{attribute 'linkalways'} 
{attribute 'no_explicit_call' := 'This FB is a CLASS and must be accessed using methods or properties'}
{attribute 'enable_dynamic_creation'}
FUNCTION_BLOCK Node_F_VN_BoxFilter EXTENDS VisionNode
VAR
	ipSrcImage : _ITcVnImage;
    ipDestImage : _ITcVnImage;
    nFilterWidth : _UDINT(1);
    nFilterHeight : _UDINT(1);
    hrPrev : _HRESULT(S_OK);
	hresult : _HRESULT(S_OK);
END_VAR

METHOD PUBLIC  Clone : I_Node
VAR
	pNode : POINTER TO Node_F_VN_BoxFilter;
END_VAR
pNode := __NEW(Node_F_VN_BoxFilter);
Clone := pNode^;
END_METHOD

METHOD FB_init : BOOL
VAR_INPUT
	bInitRetains : BOOL; // if TRUE, the retain variables are initialized (warm start / cold start)
	bInCopyCode : BOOL;  // if TRUE, the instance afterwards gets moved into the copy code (online change)
END_VAR
AddInput('ipSrcImage', ipSrcImage);
AddInput('hrPrev', hrPrev);
AddOutput('ipDestImage', ipDestImage);
AddOutput('hresult',hresult);
AddParameter('nFilterWidth', nFilterWidth);
AddParameter('nFilterHeight', nFilterHeight);
END_METHOD

METHOD PROTECTED  OnExecute : HRESULT
hresult.Value := F_VN_BoxFilter(
	ipSrcImage:= ipSrcImage.Value, 
	ipDestImage:= ipDestImage.Value, 
	nFilterWidth:= nFilterWidth.Value, 
	nFilterHeight:= nFilterHeight.Value, 
	hrPrev:= hrPrev.Value);
END_METHOD

METHOD PUBLIC PreExecutionCheck
VAR_INPUT
	Check : I_PreExecutionChecks;
END_VAR
IF FAILED(hrPrev.Value) THEN
    RETURN;
END_IF

Check.IsTrue(ipSrcImage.IsValid, 'ipSrcImage must contain an image');
Check.IsTrue((nFilterWidth.Value >= 1), 'nFilterWidth must be >= 1');
Check.IsTrue((nFilterHeight.Value >= 1), 'nFilterHeight must be >= 1');
END_METHOD

END_FUNCTION_BLOCK

(* stored: Version 1.1.0.1, ProductVersion 3.1.4024.13
   POU Node_F_VN_BoxFilter: Id {bf9b271f-fa1d-08fe-35b4-c4c2420dee84}, SpecialFunc None
   Folder Constructor: Id {dbff508c-b300-00a9-0e3b-c59e7bcd7ee3}
   Method Clone: Id {f9da4f12-ba97-09cb-0b71-f630304eb14f}
   Method FB_init: Id {ae7d20fa-99ba-0f3b-1b59-4b950d5b4120}
   Method OnExecute: Id {93a34a9e-d55e-06cc-0483-a739e5bbac47}
   Method PreExecutionCheck: Id {3b6cba54-054d-0000-1577-d02401005a0d} *)
